{attribute 'GeneratedUsingTerminal: EK1100-0000-0018'}
{attribute addProperty BoxType "EK1100-0000-0018"}
{attribute addProperty Id "Beckhoff_EPP5xxxEK1122Beckhoff_EPP5xxxEK1122_A42C9514232"}
{attribute addProperty CRC "3150968172"}
{attribute addProperty Size "232"}
TYPE Beckhoff_EPP5xxx_BBCFF56C EXTENDS EK1100_1FC0878B :
STRUCT
	{attribute addProperty Name "Beckhoff_EPP5xxxEK1122"}
	{attribute addProperty PreviousPort "Beckhoff EPP5xxx : B"}
	Beckhoff_EPP5xxxEK1122 : Beckhoff_EPP5xxxEK1122_A42C9514;
END_STRUCT
END_TYPE

(* stored: Version 1.2.0.0, ProductVersion 3.1.4024.9
   DUT Beckhoff_EPP5xxx_BBCFF56C: Id {695a17cd-330b-475b-8134-b9eca4f11260} *)
